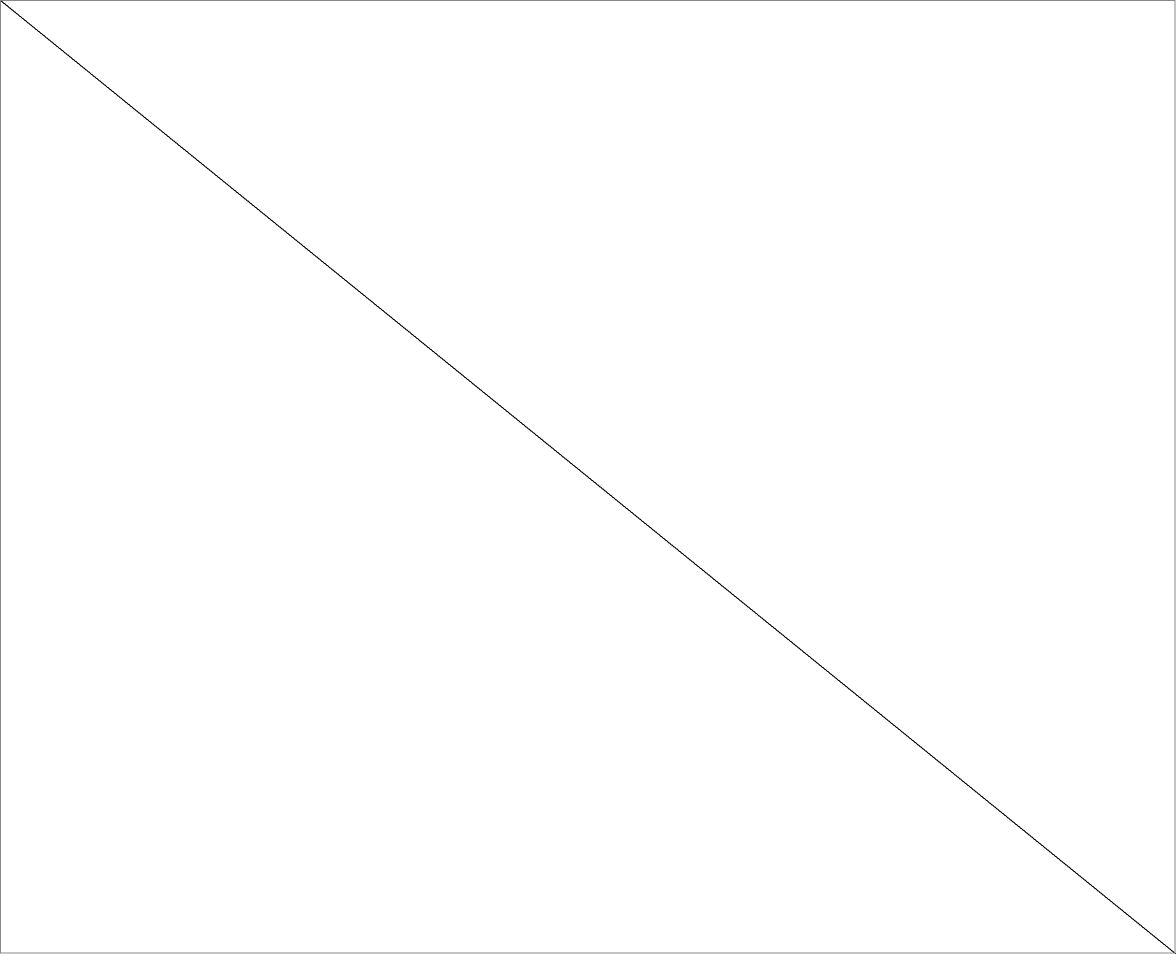
VISUALIZATION Polygon  // 1176x954
VAR_IN_OUT
	pVisu : POINTER TO ARRAY[0..999] OF VisuElems.VisuStructPoint;
	VisuLenght : INT;
END_VAR
    Polyline (0,0) (1176,954) (0,0) (0,0) (0,0)
        p1285906596: pVisu
        p3184209983: VisuLenght
END_VISUALIZATION

(* stored: Version 1.1.0.1, ProductVersion 3.1.4024.12
   Visu Polygon: Id {06e9a96e-78bb-4078-a164-82601b64cddb} *)
